{attribute addProperty BoxType "KL9900-0060"}
{attribute addProperty Id "Channel_1Channel_1B96BEED00"}
{attribute addProperty CRC "3164998640"}
{attribute addProperty SizeInBites "0"}
{attribute addProperty SizeInBytes "0"}
TYPE KL_BCA60BF0 :
STRUCT
	{attribute addProperty Name "Channel_1"}
	Channel_1 : Channel_1B96BEED;
END_STRUCT
END_TYPE

(* stored: Version 1.2.0.0, ProductVersion 3.1.4024.9
   DUT KL_BCA60BF0: Id {93432a53-a4fe-40e3-9b74-7f4ecb369db7} *)
